TYPE ST_PNInput_General :
STRUCT
	W_Control		:	WORD;
	ui_HeartBeat	:	UINT;
END_STRUCT
END_TYPE

(* stored: Version 1.1.0.1, ProductVersion 3.1.4024.12
   DUT ST_PNInput_General: Id {8077cd0e-0007-4ebb-8c06-90caa777c5f2} *)
